{attribute 'qualified_only'}
VAR_GLOBAL
	fbManualControler	: FB_ManualController ; // Default Manual control function for devices (not called implicitly) 
	bManualModeActive	: BOOL ; // System manual mode is active
END_VAR
VAR_GLOBAL CONSTANT
	nMAXDEVCOUNT		: UDINT  := 100		; // Maximum number of devices 
END_VAR

(* stored: Version 1.1.0.1, ProductVersion 3.1.4024.4
   GVL GVL_DevManual: Id {00b25fb3-c340-0c06-25e7-2c03a5c81d3c} *)
